{attribute 'GeneratedUsingTerminal: EP2809-0042-0017'}
{attribute addProperty BoxType "EP2809-0042-0017"}
{attribute addProperty Description "EP2809-0042 16 Ch. Dig. Output 24V, 0,5A, M12"}
{attribute addProperty Physics "YY"}
{attribute addProperty Id "DO_X01_Pin_4AT %Q*DO_X01_Pin_42CA91F71DO_X01_Pin_2AT %Q*DO_X01_Pin_42CA91F71DO_X02_Pin_4AT %Q*DO_X02_Pin_42CA91F71DO_X02_Pin_2AT %Q*DO_X02_Pin_42CA91F71DO_X03_Pin_4AT %Q*DO_X03_Pin_42CA91F71DO_X03_Pin_2AT %Q*DO_X03_Pin_42CA91F71DO_X04_Pin_4AT %Q*DO_X04_Pin_42CA91F71DO_X04_Pin_2AT %Q*DO_X04_Pin_42CA91F71DO_X05_Pin_4AT %Q*DO_X05_Pin_42CA91F71DO_X05_Pin_2AT %Q*DO_X05_Pin_42CA91F71DO_X06_Pin_4AT %Q*DO_X06_Pin_42CA91F71DO_X06_Pin_2AT %Q*DO_X06_Pin_42CA91F71DO_X07_Pin_4AT %Q*DO_X07_Pin_42CA91F71DO_X07_Pin_2AT %Q*DO_X07_Pin_42CA91F71DO_X08_Pin_4AT %Q*DO_X08_Pin_42CA91F71DO_X08_Pin_2AT %Q*DO_X08_Pin_42CA91F71WcStateAT %I*WcState_0B2B16F91InfoDataAT %I*InfoData_6F19DB2B2"}
{attribute addProperty CRC "2058301041"}
{attribute addProperty Size "19"}
TYPE EP2809_7AAF2E71 EXTENDS EtcSlaveBoxBase_77A0E4A7 :
STRUCT
	{attribute addProperty Name "DO_X01_Pin_4"}
	DO_X01_Pin_4 : DO_X01_Pin_42CA91F7;
	{attribute addProperty Name "DO_X01_Pin_2"}
	DO_X01_Pin_2 : DO_X01_Pin_42CA91F7;
	{attribute addProperty Name "DO_X02_Pin_4"}
	DO_X02_Pin_4 : DO_X02_Pin_42CA91F7;
	{attribute addProperty Name "DO_X02_Pin_2"}
	DO_X02_Pin_2 : DO_X02_Pin_42CA91F7;
	{attribute addProperty Name "DO_X03_Pin_4"}
	DO_X03_Pin_4 : DO_X03_Pin_42CA91F7;
	{attribute addProperty Name "DO_X03_Pin_2"}
	DO_X03_Pin_2 : DO_X03_Pin_42CA91F7;
	{attribute addProperty Name "DO_X04_Pin_4"}
	DO_X04_Pin_4 : DO_X04_Pin_42CA91F7;
	{attribute addProperty Name "DO_X04_Pin_2"}
	DO_X04_Pin_2 : DO_X04_Pin_42CA91F7;
	{attribute addProperty Name "DO_X05_Pin_4"}
	DO_X05_Pin_4 : DO_X05_Pin_42CA91F7;
	{attribute addProperty Name "DO_X05_Pin_2"}
	DO_X05_Pin_2 : DO_X05_Pin_42CA91F7;
	{attribute addProperty Name "DO_X06_Pin_4"}
	DO_X06_Pin_4 : DO_X06_Pin_42CA91F7;
	{attribute addProperty Name "DO_X06_Pin_2"}
	DO_X06_Pin_2 : DO_X06_Pin_42CA91F7;
	{attribute addProperty Name "DO_X07_Pin_4"}
	DO_X07_Pin_4 : DO_X07_Pin_42CA91F7;
	{attribute addProperty Name "DO_X07_Pin_2"}
	DO_X07_Pin_2 : DO_X07_Pin_42CA91F7;
	{attribute addProperty Name "DO_X08_Pin_4"}
	DO_X08_Pin_4 : DO_X08_Pin_42CA91F7;
	{attribute addProperty Name "DO_X08_Pin_2"}
	DO_X08_Pin_2 : DO_X08_Pin_42CA91F7;
	{attribute addProperty Name "WcState"}
	WcState : WcState_0B2B16F9;
	{attribute addProperty Name "InfoData"}
	InfoData : InfoData_6F19DB2B;
END_STRUCT
END_TYPE

(* stored: Version 1.2.0.0, ProductVersion 3.1.4024.9
   DUT EP2809_7AAF2E71: Id {91bd89a6-77f0-45d4-a44c-3442aa4a45e1} *)
